TYPE EL3204_DEV_STATUS :
    STRUCT
      
		Underrange : BOOL;
		Overrange : BOOL;
		Limit1 : BOOL;
		Limit2 : BOOL;
		Error : BOOL;
		TxPDOState : BOOL;
		TxPDOToggle : BOOL;
	
    END_STRUCT
END_TYPE

(* stored: Version 1.1.0.1, ProductVersion 3.1.4024.15
   DUT EL3204_DEV_STATUS: Id {8fc781d2-aeb7-43a7-9d35-e1d569c86329} *)
